(*$
	Returns <i>TRUE</i> if the status of the instance <b><i>this</i></b> is
	<a href="#analog_actuator_status_enum"><i>ANALOG_ACTUATOR_STATUS_INACTIVE</i></a>, 
	<i>FALSE</i> otherwise.
$*)
FUNCTION analog_actuator_is_in_range: BOOL
VAR_IN_OUT
    CONVERSION_this:	analog_actuator;	(*$ Instance to which the method applies $*)
END_VAR

IF descriptor_get_mode(CONVERSION_this.descriptor) = MODE_ABSENT
THEN
	analog_actuator_is_in_range := TRUE;
	RETURN;
END_IF

analog_actuator_is_in_range := analog_check_is_in_range(CONVERSION_this.feedback_achk);

END_FUNCTION

(* stored: Version 1.1.0.1, ProductVersion 3.1.4022.12
   POU analog_actuator_is_in_range: Id {ee9b0cef-85c7-4cdc-a898-3b88bed56ab2}, SpecialFunc None *)
